FUNCTION_BLOCK CmdAerate_HMI (* Service Interface Function Block Type *)
  (* Standard: 61499-2 *)
  (* Version 0.0, 6/7/2026, Schneider Electric, template *)
  PACKAGE SE.Nereda;
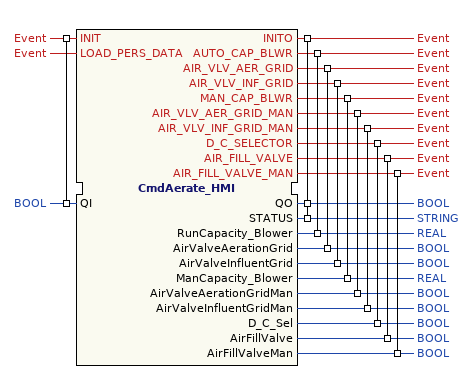
  EVENT_INPUT
    INIT WITH QI;
    LOAD_PERS_DATA;
  END_EVENT
  EVENT_OUTPUT
    INITO WITH QO, STATUS;
    AUTO_CAP_BLWR WITH RunCapacity_Blower;
    AIR_VLV_AER_GRID WITH AirValveAerationGrid;
    AIR_VLV_INF_GRID WITH AirValveInfluentGrid;
    MAN_CAP_BLWR WITH ManCapacity_Blower;
    AIR_VLV_AER_GRID_MAN WITH AirValveAerationGridMan;
    AIR_VLV_INF_GRID_MAN WITH AirValveInfluentGridMan;
    D_C_SELECTOR WITH D_C_Sel;
    AIR_FILL_VALVE WITH AirFillValve;
    AIR_FILL_VALVE_MAN WITH AirFillValveMan;
  END_EVENT
  VAR_INPUT
    QI : BOOL;
  END_VAR
  VAR_OUTPUT
    QO : BOOL; (* Event Output Qualifier *)
    STATUS : STRING; (* Service Status *)
    RunCapacity_Blower : REAL;
    AirValveAerationGrid : BOOL;
    AirValveInfluentGrid : BOOL;
    ManCapacity_Blower : REAL;
    AirValveAerationGridMan : BOOL;
    AirValveInfluentGridMan : BOOL;
    D_C_Sel : BOOL;
    AirFillValve : BOOL;
    AirFillValveMan : BOOL;
  END_VAR
  SERVICE /
    SEQUENCE 
    END_SEQUENCE
  END_SERVICE
END_FUNCTION_BLOCK
